FUNCTION_BLOCK AtvPowerCalculator (* Basic Function Block Type *)
  (* Standard: 61499-2 *)
  (* Version 0.0, 8/23/2024, SESA713705, Schneider Electric, Template *)
  PACKAGE SE.Nereda;
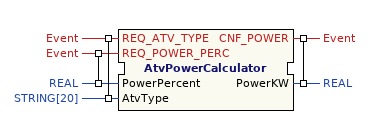
  EVENT_INPUT
    REQ_ATV_TYPE WITH AtvType;
    REQ_POWER_PERC WITH PowerPercent;
  END_EVENT
  EVENT_OUTPUT
    CNF_POWER WITH PowerKW;
  END_EVENT
  VAR_INPUT
    PowerPercent : REAL;
    AtvType : STRING[20];
  END_VAR
  VAR_OUTPUT
    PowerKW : REAL;
  END_VAR
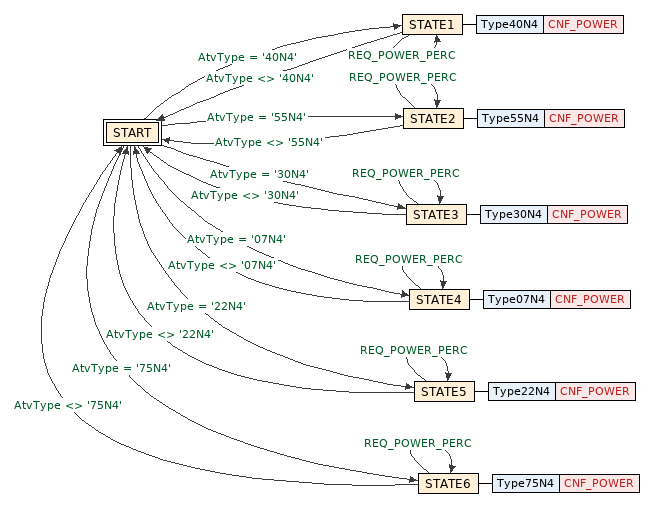
  EC_STATES
    START; (* Initial State *)
    STATE1 : Type40N4 -> CNF_POWER;
    STATE2 : Type55N4 -> CNF_POWER;
    STATE3 : Type30N4 -> CNF_POWER;
    STATE4 : Type07N4 -> CNF_POWER;
    STATE5 : Type22N4 -> CNF_POWER;
    STATE6 : Type75N4 -> CNF_POWER;
  END_STATES
  EC_TRANSITIONS
    START TO STATE1 := AtvType = '40N4';
    STATE1 TO START := AtvType <> '40N4';
    START TO STATE2 := AtvType = '55N4';
    STATE2 TO START := AtvType <> '55N4';
    START TO STATE3 := AtvType = '30N4';
    STATE3 TO START := AtvType <> '30N4';
    START TO STATE4 := AtvType = '07N4';
    STATE4 TO START := AtvType <> '07N4';
    START TO STATE5 := AtvType = '22N4';
    STATE5 TO START := AtvType <> '22N4';
    START TO STATE6 := AtvType = '75N4';
    STATE6 TO START := AtvType <> '75N4';
    STATE1 TO STATE1 := REQ_POWER_PERC;
    STATE2 TO STATE2 := REQ_POWER_PERC;
    STATE3 TO STATE3 := REQ_POWER_PERC;
    STATE4 TO STATE4 := REQ_POWER_PERC;
    STATE5 TO STATE5 := REQ_POWER_PERC;
    STATE6 TO STATE6 := REQ_POWER_PERC;
  END_TRANSITIONS
  ALGORITHM Type40N4 IN ST:
;
PowerKW := (PowerPercent/100) * 2.8;
  END_ALGORITHM
  ALGORITHM Type55N4 IN ST:
;
PowerKW := (PowerPercent/100) * 4;
  END_ALGORITHM
  ALGORITHM Type30N4 IN ST:
;
PowerKW := (PowerPercent/100) * 1.5;
  END_ALGORITHM
  ALGORITHM Type07N4 IN ST:
;
PowerKW := (PowerPercent/100) * 0.37;
  END_ALGORITHM
  ALGORITHM Type22N4 IN ST:
;
PowerKW := (PowerPercent/100) * 1.8;
  END_ALGORITHM
  ALGORITHM Type75N4 IN ST:
;
PowerKW := (PowerPercent/100) * 6;
  END_ALGORITHM
END_FUNCTION_BLOCK
